(* IEC 61131-3 sources: Std_PalletMover/Class/BasicHardwareInterface, 1 file *)

(* ---- BasicHardwareInterface.st ---- *)
(*!
<Class
	Name               = "BasicHardwareInterface"
	Revision           = "0.0"
	RealtimeTask       = "false"
	CyclicTask         = "false"
	BackgroundTask     = "false"
	Sigmatek           = "false"
	OSInterface        = "false"
	HighPriority       = "false"
	Automatic          = "false"
	UpdateMode         = "Prescan"
	SharedCommandTable = "true"
	Objectsize         = "(810,120)">
	<Channels>
		<Client Name="LiftAnalogHeight" Required="true" Internal="false"/>
		<Client Name="LiftSensorDriveHeight" Required="true" Internal="false"/>
		<Client Name="LiftSensorMaxHeight" Required="true" Internal="false"/>
		<Client Name="LiftSensorMinHeight" Required="true" Internal="false"/>
	</Channels>
	<Network Name="BasicHardwareInterface">
		<!-- List of Components in this network -->
		<Components>
			<Object
				Name       = "_base"
				Class      = "HardwareBase"
				Position   = "(218,120)"
				Visualized = "false">
				<Channels>
					<Server Name="ToObject"/>
					<Client Name="op_LogData"/>
					<Client Name="p_NextObject"/>
				</Channels>
			</Object>
		</Components>
		<Comments>
		</Comments>
		<!-- List of Connections in this network -->
		<Connections>
			<Connection Source="this.ToObject" Destination="_base.ToObject" Vertices="(976,210),(804,210),"/>
		</Connections>
		<!-- Headerfiles -->
		<Options>
		</Options>
	</Network>
</Class>
*)
#pragma using HardwareBase

BasicHardwareInterface : CLASS
: HardwareBase
  //Servers:
  //Clients:
	LiftSensorMaxHeight 	: CltCh_DINT;
	LiftSensorMinHeight 	: CltCh_DINT;
	LiftSensorDriveHeight 	: CltCh_DINT;
	LiftAnalogHeight 	: CltCh_DINT;
  //Variables:
  //Functions:
  //Tables:
	FUNCTION @STD
		VAR_OUTPUT
			ret_code	: CONFSTATES;
		END_VAR;
	FUNCTION GLOBAL TAB @CT_;
END_CLASS;
